FUNCTION_BLOCK Eigenvector2x2 (* Composite FB wrapping other FBs *)
  (* Standard: 61499-2; Description: Part of ellipse fitting method, to find eigenvalue. This block are specifically in use of ellipse fitting method, which doesn't generally exported. *)
  (* Version 1.0, 2020-08-19, Candra Wardaya, UGM *)
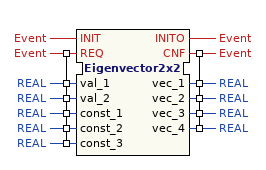
  EVENT_INPUT
    INIT; (* Initialization Request *)
    REQ WITH const_1, const_2, const_3, val_1, val_2; (* Normal Execution Request *)
  END_EVENT
  EVENT_OUTPUT
    INITO; (* Initialization Confirm *)
    CNF WITH vec_1, vec_2, vec_3, vec_4; (* Execution Confirmation *)
  END_EVENT
  VAR_INPUT
    val_1 : REAL;
    val_2 : REAL;
    const_1 : REAL; (* Single Real Input *)
    const_2 : REAL; (* Single Real Input *)
    const_3 : REAL; (* Single Real Input *)
  END_VAR
  VAR_OUTPUT
    vec_1 : REAL; (* Single Real Output *)
    vec_2 : REAL;
    vec_3 : REAL;
    vec_4 : REAL;
  END_VAR
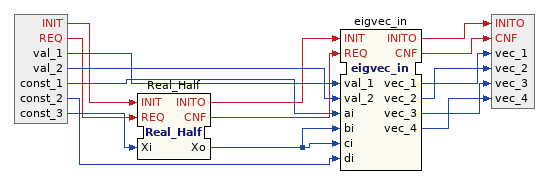
  FBS
    Real_Half : Real_Half;
    eigvec_in : eigvec_in;
  END_FBS
  EVENT_CONNECTIONS
    REQ TO Real_Half.REQ;
    INIT TO Real_Half.INIT;
    Real_Half.INITO TO eigvec_in.INIT;
    Real_Half.CNF TO eigvec_in.REQ;
    eigvec_in.INITO TO INITO;
    eigvec_in.CNF TO CNF;
  END_CONNECTIONS
  DATA_CONNECTIONS
    const_3 TO Real_Half.Xi;
    val_1 TO eigvec_in.val_1;
    val_2 TO eigvec_in.val_2;
    const_1 TO eigvec_in.ai;
    const_2 TO eigvec_in.di;
    Real_Half.Xo TO eigvec_in.bi;
    Real_Half.Xo TO eigvec_in.ci;
    eigvec_in.vec_1 TO vec_1;
    eigvec_in.vec_2 TO vec_2;
    eigvec_in.vec_3 TO vec_3;
    eigvec_in.vec_4 TO vec_4;
  END_CONNECTIONS
END_FUNCTION_BLOCK
